{attribute 'linkalways'} 
{attribute 'no_explicit_call' := 'This FB is a CLASS and must be accessed using methods or properties'}
{attribute 'enable_dynamic_creation'}
FUNCTION_BLOCK Node_F_VN_DrawCircularArc EXTENDS VisionNode
VAR
    stCircularArc : _TcVnCircularArc;
    ipDestImage : _ITcVnImage;
    aColor : _TcVnVector4_LREAL;
    nThickness : _DINT(1);
    hrPrev : _HRESULT(S_OK);
	hresult : _HRESULT(S_OK);
END_VAR

METHOD PUBLIC  Clone : I_Node
VAR
	pNode : POINTER TO Node_F_VN_DrawCircularArc;
END_VAR
pNode := __NEW(Node_F_VN_DrawCircularArc);
Clone := pNode^;
END_METHOD

METHOD FB_init : BOOL
VAR_INPUT
	bInitRetains : BOOL; // if TRUE, the retain variables are initialized (warm start / cold start)
	bInCopyCode : BOOL;  // if TRUE, the instance afterwards gets moved into the copy code (online change)
END_VAR
AddInput('stCircularArc', stCircularArc);
AddInput('ipDestImage', ipDestImage);
AddInput('aColor', aColor);
AddParameter('nThickness', nThickness);
AddInput('hrPrev', hrPrev);
AddOutput('ipDestImage', ipDestImage);
AddOutput('hresult',hresult);
END_METHOD

METHOD PROTECTED OnExecute
hresult.Value := F_VN_DrawCircularArc(
    stCircularArc := stCircularArc.Value,
	ipDestImage := ipDestImage.Value,
    aColor := aColor.Value,
    nThickness := nThickness.Value,
	hrPrev:= hrPrev.Value);
END_METHOD

METHOD PUBLIC PreExecutionCheck
VAR_INPUT
	Check : I_PreExecutionChecks;
END_VAR
Check.IsTrue(ipDestImage.IsValid, 'ipDestImage must contain an image');
Check.IsTrue(nThickness.Value <> 0, 'nThickness must be non-zero');
END_METHOD

END_FUNCTION_BLOCK

(* stored: Version 1.1.0.1, ProductVersion 3.1.4024.15
   POU Node_F_VN_DrawCircularArc: Id {e0caeaa2-21d3-02e7-3e41-6182e5619c9a}, SpecialFunc None
   Folder Constructor: Id {712e5317-d1b6-0a81-38ab-47e6219ca87c}
   Method Clone: Id {267baf55-e47a-00d2-3e9d-cd300dfd8e18}
   Method FB_init: Id {d167c0da-f0f2-09e6-1b0d-62b5cb3897db}
   Method OnExecute: Id {1da798e9-1408-0151-2524-4a41e0e7b6ce}
   Method PreExecutionCheck: Id {2170627d-e9c8-0f1b-3b75-80dd33e31f92} *)
